(* PLC project Unnamed, Unknown Unnamed 1 *)
(* stored: creationDateTime 2025-10-24T14:34:45, modificationDateTime 2025-10-27T19:28:33 *)

PROGRAM program0
  VAR
    StartButton : BOOL;
    StopButton : BOOL;
    Process : BOOL;
    RoomHot : BOOL;
    MeasuredTemp : INT;
    ThresholdTemp : INT := 21;
    AirCon : BOOL;
  END_VAR

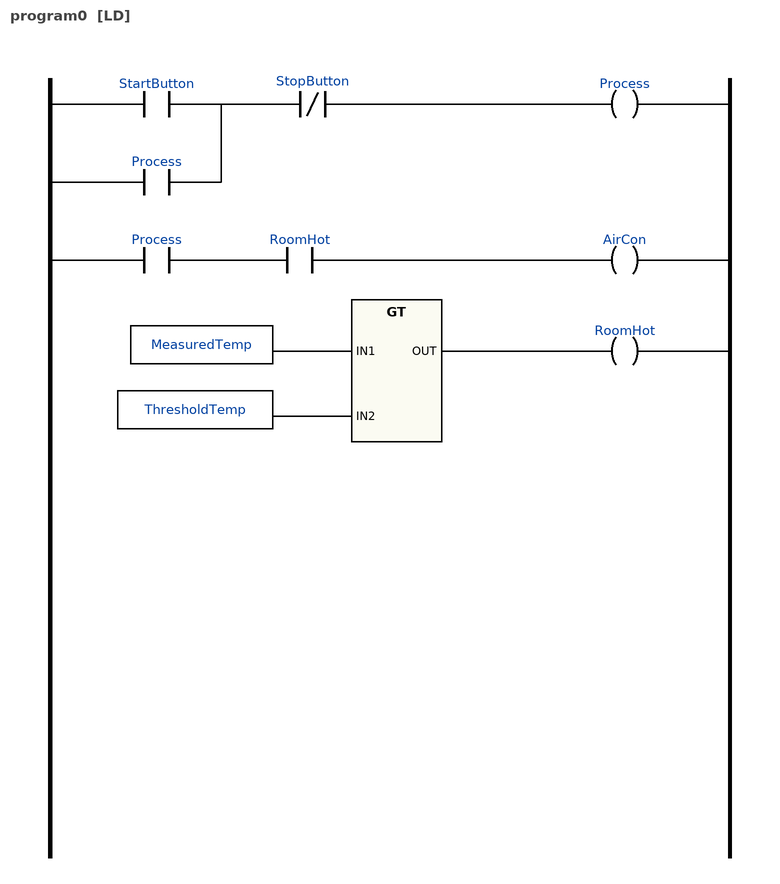
(* LD diagram, written out as Structured Text *)
Process := (StartButton OR Process) AND NOT StopButton;
AirCon := Process AND RoomHot;
RoomHot := MeasuredTemp > ThresholdTemp;
END_PROGRAM

CONFIGURATION Config0
  RESOURCE Res0 ON PLC
    TASK task0(INTERVAL := T#20ms, PRIORITY := 0);
    PROGRAM instance0 WITH task0 : program0;
  END_RESOURCE
END_CONFIGURATION
